// TIA Portal V18 export
// export: Created 2026-06-11T17:34:54.6885639Z, ExportSetting WithDefaults, DisplayName Totally Integrated Automation Portal, DisplayVersion V18, DisplayName TIA Portal Openness, DisplayVersion V18, DisplayName TIA Portal Version Control Interface, DisplayVersion V18, DisplayName STEP 7 Professional, DisplayVersion V18, DisplayName STEP 7 Safety, DisplayVersion V18, DisplayName WinCC Professional, DisplayVersion V18
Screen "Login/out"  1920x1080, Number=1
  ScreenLayer 
    GraphicView "Graphic view_1" at 0,0 size 1920x1080  Picture=backgroundadmin
    Button "Btn_Login" at 780,369 size 397x64  Mode=Text, StyleItem=Button, TextOff="ĐĂNG NHẬP (LOGIN)", TextOn="Text"
      VisibilityAnimation "VisibilityAnimation"
        tag Logged_In
      on Click: ShowLogonDialog()
    Button "Btn_Enter_System" at 781,461 size 398x61  Mode=Text, StyleItem=Button, TextOff="VÀO HỆ THỐNG (SCADA)", TextOn="Text"
      VisibilityAnimation "VisibilityAnimation"  RangeEnd=99, RangeStart=1
        tag Logged_In
      on Click: ActivateScreen(Screen name := Screen_2, Object number := 0)
    Button "Btn_Logout" at 780,561 size 401x65  Mode=Text, StyleItem=Button, TextOff="ĐĂNG XUẤT (LOGOFF)", TextOn="Text"
      VisibilityAnimation "VisibilityAnimation"  RangeEnd=99, RangeStart=1
        tag Logged_In
      on Click: Logoff()
    Button "Btn_Exit" at 781,649 size 402x51  Mode=Text, StyleItem=Button, TextOff="THOÁT HỆ THỐNG (EXIT)", TextOn="Text"
      on Click: StopRuntime(Mode := 0)
